{attribute 'linkalways'} 
{attribute 'no_explicit_call' := 'This FB is a CLASS and must be accessed using methods or properties'}
{attribute 'enable_dynamic_creation'}
FUNCTION_BLOCK FINAL MOD_ULINT EXTENDS Node
VAR
	in1 : _ULINT(0);
	in2 : _ULINT(0);
	out : _ULINT(0);
END_VAR

METHOD PUBLIC Clone : I_Node
VAR
	pNode : POINTER TO MOD_ULINT;
END_VAR
pNode := __NEW(MOD_ULINT);
Clone := pNode^;
END_METHOD

METHOD FB_init : BOOL
VAR_INPUT
	bInitRetains : BOOL; // if TRUE, the retain variables are initialized (warm start / cold start)
	bInCopyCode : BOOL;  // if TRUE, the instance afterwards gets moved into the copy code (online change)
END_VAR
AddInput('in1',THIS^.in1);
AddInput('in2',THIS^.in2);
AddOutput('out', THIS^.out);
END_METHOD

METHOD PROTECTED OnExecute
VAR
END_VAR
out.Value := in1.Value MOD in2.Value;
END_METHOD

END_FUNCTION_BLOCK

(* stored: Version 1.1.0.1, ProductVersion 3.1.4024.15
   POU MOD_ULINT: Id {41cd86a1-fa1c-47bc-86a8-5a82c3859181}, SpecialFunc None
   Folder Constructor: Id {2e3baaa8-b00c-4d82-b514-9cb97d94f90d}
   Method Clone: Id {cc7569a3-1e99-4956-b74d-d187199b7743}
   Method FB_init: Id {b0c8525b-e33c-48f0-a8dc-a40f7746573d}
   Method OnExecute: Id {883cb557-c207-4d7f-9308-4f57ee76119a} *)
